{attribute 'linkalways'} 
{attribute 'no_explicit_call' := 'This FB is a CLASS and must be accessed using methods or properties'}
{attribute 'enable_dynamic_creation'}
FUNCTION_BLOCK _ETcVnBarcodeSearchDirection EXTENDS EnumDatatypeBase
VAR
	localData : ETcVnBarcodeSearchDirection;
	activeData : REFERENCE TO ETcVnBarcodeSearchDirection;
	enumBaseDatatype : _UDINT(localData);
END_VAR

METHOD PRIVATE AddLocalEnumeration
VAR_INPUT
	Enumeration : T_MAXSTRING;
	Value : ETcVnBarcodeSearchDirection;
END_VAR
AddEnumeration(Enumeration, Value);
END_METHOD

PROPERTY PUBLIC Address : PVOID
GET
Address := ADR(activeData);
END_GET
END_PROPERTY

METHOD PUBLIC ClearReference
VAR_INPUT
END_VAR
activeData REF= localData;
SetBaseDatatypeReference();
END_METHOD

METHOD PUBLIC Clone : I_Datatype
VAR
    pClone : POINTER TO _ETcVnBarcodeSearchDirection;
END_VAR
pClone := __NEW(_ETcVnBarcodeSearchDirection(InitialValue := Value));
Clone := pClone^;
END_METHOD

METHOD FB_init : BOOL
VAR_INPUT
	bInitRetains : BOOL; // if TRUE, the retain variables are initialized (warm start / cold start)
	bInCopyCode : BOOL;  // if TRUE, the instance afterwards gets moved into the copy code (online change)
	InitialValue : ETcVnBarcodeSearchDirection;
END_VAR
localData := InitialValue;
AddBaseDatatype(enumBaseDatatype);
ClearReference();

AddLocalEnumeration('TCVN_BSD_ANY', ETcVnBarcodeSearchDirection.TCVN_BSD_ANY);
AddLocalEnumeration('TCVN_BSD_HORIZONTAL', ETcVnBarcodeSearchDirection.TCVN_BSD_HORIZONTAL);
AddLocalEnumeration('TCVN_BSD_VERTICAL', ETcVnBarcodeSearchDirection.TCVN_BSD_VERTICAL);
END_METHOD

PROPERTY PUBLIC Identifier : T_MAXSTRING
GET
Identifier := 'ETcVnBarcodeSearchDirection';
END_GET
END_PROPERTY

METHOD IsEnumeratorValueEqual : BOOL
VAR_INPUT
	Enumerator : I_KeyValueForwardEnumerator;
END_VAR
VAR
	storedValue : ETcVnBarcodeSearchDirection;
END_VAR
IF NOT Enumerator.TryGet(storedValue) THEN
	RETURN;
END_IF

IsEnumeratorValueEqual := storedValue = activeData;
END_METHOD

METHOD PUBLIC MakeReferenceTo
VAR_INPUT
	ReferenceTarget : REFERENCE TO ETcVnBarcodeSearchDirection;
END_VAR
activeData REF= ReferenceTarget;
SetBaseDatatypeReference();
END_METHOD

METHOD PROTECTED SetBaseDatatypeReference
VAR_INPUT
END_VAR
enumBaseDatatype.MakeReferenceTo(activeData);
END_METHOD

PROPERTY PUBLIC Size : UDINT
GET
Size := SIZEOF(activeData);
END_GET
END_PROPERTY

METHOD TryMakeReferenceTo : BOOL
VAR_INPUT
	Target : I_Datatype;
END_VAR
VAR
	targetAsEnum : I_EnumDatatype;
	pTargetData : POINTER TO ETcVnBarcodeSearchDirection;
END_VAR
IF NOT Target.TryResolveAsEnumDatatype(targetAsEnum) THEN
	RETURN;
END_IF

IF targetAsEnum.Identifier <> Identifier THEN
	RETURN;
END_IF

pTargetData := Target.Address;
activeData REF= pTargetData^;
SetBaseDatatypeReference();
TryMakeReferenceTo := TRUE;
END_METHOD

PROPERTY PUBLIC Value : ETcVnBarcodeSearchDirection
GET
Value := activeData;
END_GET
SET
activeData := Value;
END_SET
END_PROPERTY

END_FUNCTION_BLOCK

(* stored: Version 1.1.0.1, ProductVersion 3.1.4024.13
   POU _ETcVnBarcodeSearchDirection: Id {c24a8b56-f5e4-4192-99bc-66b6387fc46d}, SpecialFunc None
   Folder Core: Id {b9530c9f-d6dd-0e8b-35b1-d3cdd4e029c9}
   Folder Protected: Id {a63cfb06-6e87-0513-0f75-36a451a70474}
   Folder Customize: Id {d25fbda5-dac5-09e2-247e-d51404d13250}
   Folder Constructor: Id {df340227-9802-47ba-a3a4-361915b5c2bb}
   Folder Private: Id {4891bd97-d116-4f6c-82fa-6b1660120486}
   Folder Protected: Id {0a8c21ad-7611-4215-94ea-4ea443e541a9}
   Method AddLocalEnumeration: Id {bf34e210-580c-487a-984f-16c23ddee6a8}
   Property Address: Id {8d8d925d-801c-0577-2731-fe194c03db35}
   Get Get: Id {f225d95c-1989-0851-114e-6381685fc714}
   Method ClearReference: Id {5cc9fbc0-1032-0813-0ca7-906e9dfcbd8b}
   Method Clone: Id {d89366ea-fd23-4f0e-9f1d-e1b733772e0f}
   Method FB_init: Id {9aff6333-07ce-41c7-910e-5d39fc6e4eb6}
   Property Identifier: Id {a25247b1-0c11-4382-a831-2ed84d0613a1}
   Get Get: Id {5a75609d-f279-4f19-92d6-954979ea0a72}
   Method IsEnumeratorValueEqual: Id {cc3fbc28-b221-4f05-8da0-2b383813cee2}
   Method MakeReferenceTo: Id {df8194e9-02f2-4032-8bb5-44df1fc6d33f}
   Method SetBaseDatatypeReference: Id {1ebf78db-6320-09a1-176f-10f1906a937b}
   Property Size: Id {c9dcf8a9-0145-0459-1112-f2c152f3b3cf}
   Get Get: Id {5839793e-4fc5-081b-122d-a5643ed7d539}
   Method TryMakeReferenceTo: Id {96d78722-eb17-48eb-a9d1-6b497c3fb49f}
   Property Value: Id {92786066-2b66-4a79-b502-4f14523308b8}
   Get Get: Id {275cc093-7f62-40e9-874d-2e32bb953173}
   Set Set: Id {8c987d80-87e5-42b9-a61d-50cae82d497c} *)
